FUNCTION_BLOCK FB_Direction
VAR_INPUT
	bAutomat:BOOL;
	bManual:BOOL;
	bDirectOn :BOOL;
	bReverseOn:BOOL;
	bButtReverse:BOOL;
END_VAR
VAR_OUTPUT
	bSwitchOnDirect:BOOL:=FALSE;
	bSwitchOnReverse:BOOL:=FALSE;
END_VAR
VAR
	bModeDirect:BOOL;
	bModeReverse:BOOL;
	fbPulsButt:R_TRIG;
	fbDelayOnDirect:TON;
	fbDelayOffDirect:TON;
END_VAR


fbDelayOnDirect(IN:=NOT bReverseOn, PT:=T#1S);

IF (bManual OR bAutomat) AND fbDelayOnDirect.Q(*NOT bReverseOn*) THEN
	bSwitchOnDirect:=TRUE;
END_IF
IF NOT (bManual OR bAutomat) THEN 
	bSwitchOnDirect:=FALSE;
END_IF

 fbDelayOffDirect(IN:=NOT bDirectOn, PT:=T#1S);   

fbPulsButt(CLK:=bButtReverse  );
IF fbPulsButt.Q AND bManual AND NOT bModeReverse  THEN
bModeReverse:=TRUE;
END_IF
IF bModeReverse THEN
	bSwitchOnDirect:=FALSE;
	IF NOT bSwitchOnDirect AND (*NOT bDirectOn*)fbDelayOffDirect.Q THEN
		bSwitchOnReverse:=TRUE;
	END_IF
END_IF

IF fbPulsButt.Q AND bReverseOn  THEN
	bSwitchOnReverse:=FALSE;
	bModeReverse :=FALSE;
END_IF

END_FUNCTION_BLOCK

(* stored: Version 1.1.0.1, ProductVersion 3.1.4024.4
   POU FB_Direction: Id {e3e4167a-608f-4854-a9cd-c32589cd5b27}, SpecialFunc None *)
